# EPICS substitutions: src/makeBaseApp/top/pcdsModuleLib/Db/archive__APPNAME_.substitutions
#
# _APPNAME_ archive substitutions file
#

# Generate _APPNAME_ archive file
#	Macros:
#		TODO:	List here any macros used in the template
#				Note which ones have defaults.
file archive__APPNAME_.template
{
	{
		# Hack till msi supports empty substitutions
		IOC		=	$(IOC),
	}
}
